// Block: IPC_Com_Channel_LOG_ENERGIA

DATA_BLOCK IPC_Com_Channel_LOG_ENERGIA
VERSION : 0.1
   NON_RETAIN
   VAR
      SEND : Struct
         ack : DInt;
         msg : IPC_Msg_Generico;
      END_STRUCT;
   END_VAR

BEGIN
   // No initialization required
END_DATA_BLOCK
